// TIA Portal V20 export
VAR_GLOBAL   // PLC tag table "LGR_Const_LayoutType"
END_VAR
VAR_GLOBAL CONSTANT   // user constants
   LAYOUT_RND : SInt := 0;
   LAYOUT_INSFECTION_1 : SInt := 11;
   LAYOUT_TBR_INBOUND_1 : SInt := 101;
   LAYOUT_INSFECTION_2 : SInt := 21;
   LAYOUT_INBOUND_2 : SInt := 22;
   LAYOUT_INBOUND_1 : SInt := 12;
   LAYOUT_OUTBOUND_RETURN_1 : SInt := 31;
   LAYOUT_OUTBOUND_1 : SInt := 41;
   LAYOUT_OUTBOUND_2 : SInt := 51;
   LAYOUT_OUTBOUND_3 : SInt := 61;
END_VAR
